Staubli VAL3: MotionCmdVel.dtx

public num nSequence
public num nVelCmd[6]
public num nCmdType
